FUNCTION_BLOCK FB_ModeSelector
VAR_INPUT
	bControlBox : BOOL;
END_VAR
VAR_OUTPUT
END_VAR
VAR
	fbModeVisualization : FB_ModeVisualization;
	fbModeControlBox : FB_ModeControlBox;
	fbMode : I_Mode := fbModeVisualization;
END_VAR

IF NOT(bControlBox) THEN 
	fbMode := fbModeVisualization;
	IF NOT(HMI.bOn) THEN
			fbMode.Off(TRUE); 
			fbMode.Manual(FALSE); 
			fbMode.Auto(FALSE); 
	ELSIF HMI.bOn AND NOT(HMI.bAuto) THEN
			fbMode.Off(FALSE); 
			fbMode.Manual(TRUE); 
			fbMode.Auto(FALSE); 
	ELSIF HMI.bOn AND HMI.bAuto THEN	
			fbMode.Off(FALSE); 
			fbMode.Manual(FALSE); 
			fbMode.Auto(TRUE); 
	ELSE	
			fbMode.Off(FALSE); 
			fbMode.Manual(FALSE); 
			fbMode.Auto(FALSE); 	
	END_IF
	
	
ELSE	  
	fbMode := fbModeControlBox;
	IF NOT(Inputs.bManualMode) AND NOT(Inputs.bAutoMode) THEN
			fbMode.Off(TRUE); 
			fbMode.Manual(FALSE); 
			fbMode.Auto(FALSE); 
	ELSIF Inputs.bManualMode AND NOT(Inputs.bAutoMode) THEN
			fbMode.Off(FALSE); 
			fbMode.Manual(TRUE); 
			fbMode.Auto(FALSE); 
	ELSIF NOT(Inputs.bManualMode) AND Inputs.bAutoMode THEN	
			fbMode.Off(FALSE); 
			fbMode.Manual(FALSE); 
			fbMode.Auto(TRUE); 
	ELSE	
			fbMode.Off(FALSE); 
			fbMode.Manual(FALSE); 
			fbMode.Auto(FALSE); 	
	END_IF
	
END_IF

END_FUNCTION_BLOCK

(* stored: Version 1.1.0.1, ProductVersion 3.1.4024.10
   POU FB_ModeSelector: Id {e22295b4-f0de-4c1e-b830-372a1bffee19}, SpecialFunc None *)
